// TIA Portal V21 export
// export: Created 2026-09-06T16:35:00Z, ExportSetting WithDefaults
FUNCTION "FC_LinhaCompactador_LAD" : Void   // FC21, LAD
{ S7_Optimized_Access := 'TRUE' }
VERSION : 0.1
// Visualizacao LAD da logica principal. A sequencia temporizada executavel continua em FB_LinhaCompactador.
// stored: AutoNumber true, SetENOAutomatically false
BEGIN

REGION Network 1: FC1 - OK_SISTEMA: cadeia geral de seguranca
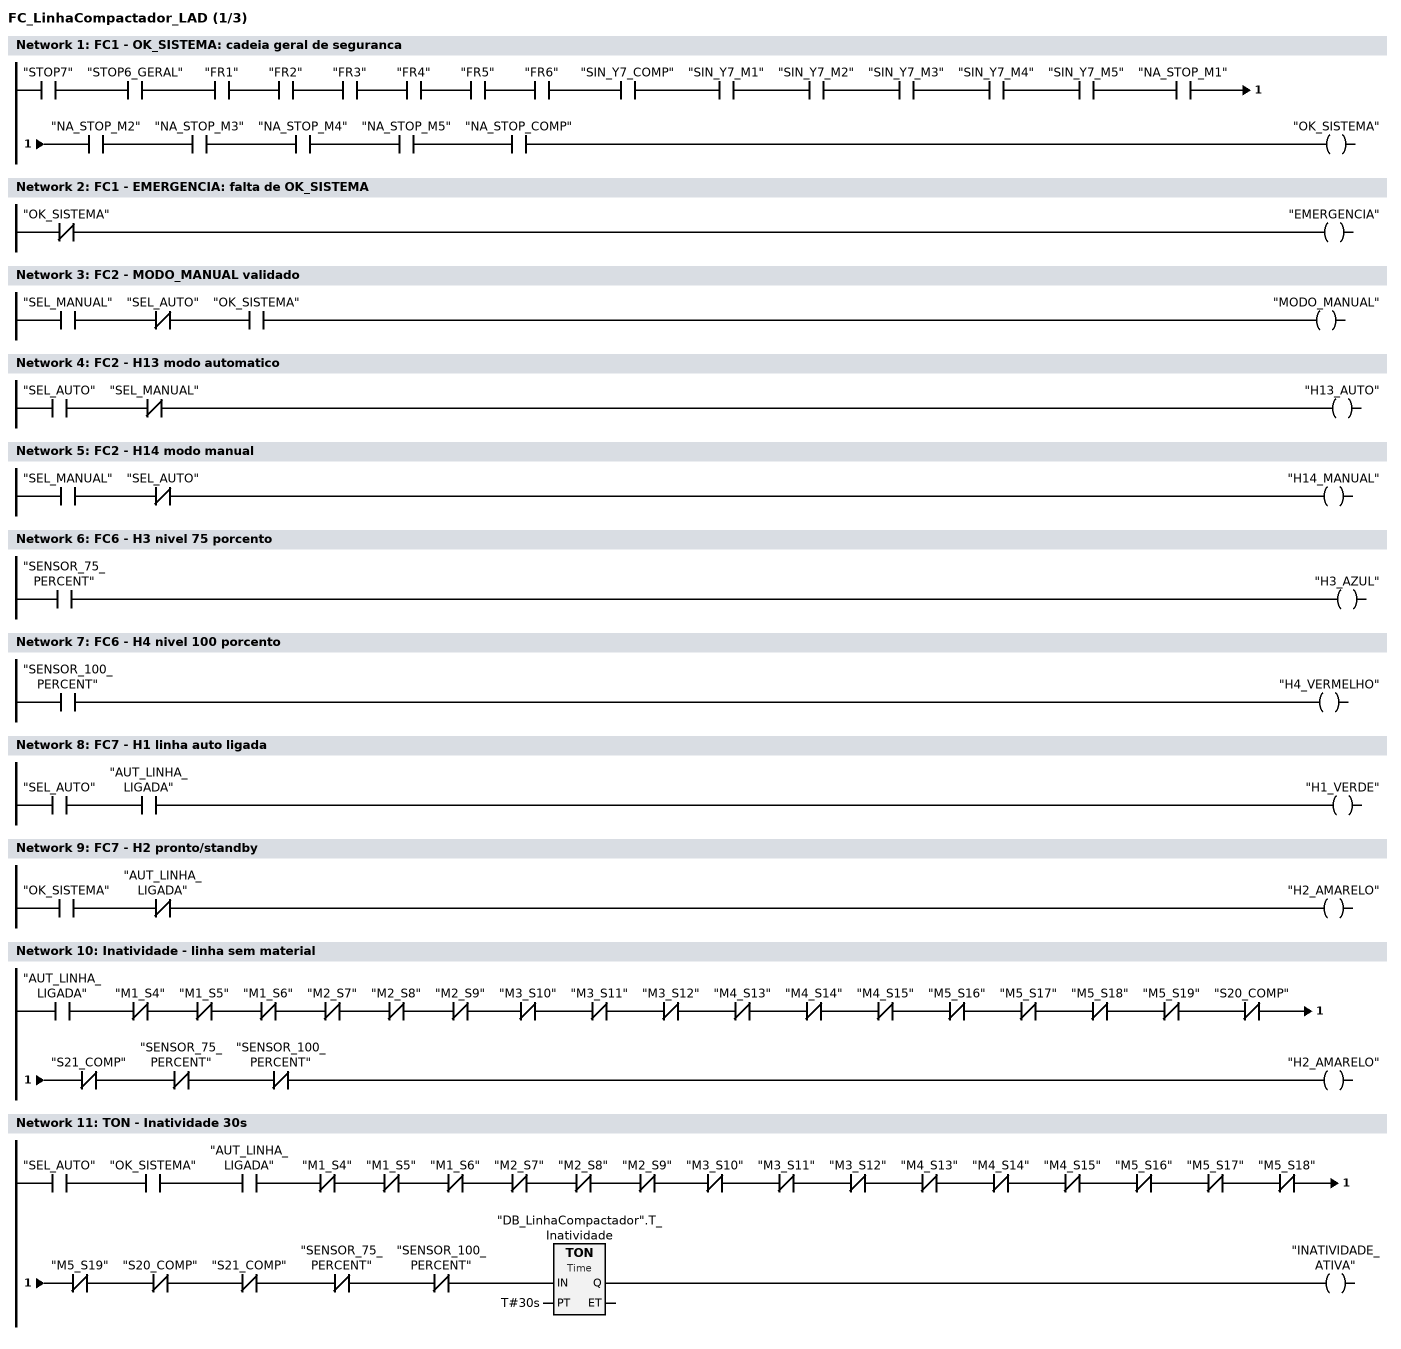
   RUNG wire#powerrail
      Contact( "STOP7" )
      Contact( "STOP6_GERAL" )
      Contact( "FR1" )
      Contact( "FR2" )
      Contact( "FR3" )
      Contact( "FR4" )
      Contact( "FR5" )
      Contact( "FR6" )
      Contact( "SIN_Y7_COMP" )
      Contact( "SIN_Y7_M1" )
      Contact( "SIN_Y7_M2" )
      Contact( "SIN_Y7_M3" )
      Contact( "SIN_Y7_M4" )
      Contact( "SIN_Y7_M5" )
      Contact( "NA_STOP_M1" )
      Contact( "NA_STOP_M2" )
      Contact( "NA_STOP_M3" )
      Contact( "NA_STOP_M4" )
      Contact( "NA_STOP_M5" )
      Contact( "NA_STOP_COMP" )
      Coil( "OK_SISTEMA" )
   END_RUNG
   // the same network as SCL:
   "OK_SISTEMA" := "STOP7" AND "STOP6_GERAL" AND "FR1" AND "FR2" AND "FR3" AND "FR4" AND "FR5" AND "FR6" AND "SIN_Y7_COMP" AND "SIN_Y7_M1" AND "SIN_Y7_M2" AND "SIN_Y7_M3" AND "SIN_Y7_M4" AND "SIN_Y7_M5" AND "NA_STOP_M1" AND "NA_STOP_M2" AND "NA_STOP_M3" AND "NA_STOP_M4" AND "NA_STOP_M5" AND "NA_STOP_COMP";
END_REGION

REGION Network 2: FC1 - EMERGENCIA: falta de OK_SISTEMA
   RUNG wire#powerrail
      I_Contact( "OK_SISTEMA" )
      Coil( "EMERGENCIA" )
   END_RUNG
   // the same network as SCL:
   "EMERGENCIA" := NOT "OK_SISTEMA";
END_REGION

REGION Network 3: FC2 - MODO_MANUAL validado
   RUNG wire#powerrail
      Contact( "SEL_MANUAL" )
      I_Contact( "SEL_AUTO" )
      Contact( "OK_SISTEMA" )
      Coil( "MODO_MANUAL" )
   END_RUNG
   // the same network as SCL:
   "MODO_MANUAL" := "SEL_MANUAL" AND NOT "SEL_AUTO" AND "OK_SISTEMA";
END_REGION

REGION Network 4: FC2 - H13 modo automatico
   RUNG wire#powerrail
      Contact( "SEL_AUTO" )
      I_Contact( "SEL_MANUAL" )
      Coil( "H13_AUTO" )
   END_RUNG
   // the same network as SCL:
   "H13_AUTO" := "SEL_AUTO" AND NOT "SEL_MANUAL";
END_REGION

REGION Network 5: FC2 - H14 modo manual
   RUNG wire#powerrail
      Contact( "SEL_MANUAL" )
      I_Contact( "SEL_AUTO" )
      Coil( "H14_MANUAL" )
   END_RUNG
   // the same network as SCL:
   "H14_MANUAL" := "SEL_MANUAL" AND NOT "SEL_AUTO";
END_REGION

REGION Network 6: FC6 - H3 nivel 75 porcento
   RUNG wire#powerrail
      Contact( "SENSOR_75_PERCENT" )
      Coil( "H3_AZUL" )
   END_RUNG
   // the same network as SCL:
   "H3_AZUL" := "SENSOR_75_PERCENT";
END_REGION

REGION Network 7: FC6 - H4 nivel 100 porcento
   RUNG wire#powerrail
      Contact( "SENSOR_100_PERCENT" )
      Coil( "H4_VERMELHO" )
   END_RUNG
   // the same network as SCL:
   "H4_VERMELHO" := "SENSOR_100_PERCENT";
END_REGION

REGION Network 8: FC7 - H1 linha auto ligada
   RUNG wire#powerrail
      Contact( "SEL_AUTO" )
      Contact( "AUT_LINHA_LIGADA" )
      Coil( "H1_VERDE" )
   END_RUNG
   // the same network as SCL:
   "H1_VERDE" := "SEL_AUTO" AND "AUT_LINHA_LIGADA";
END_REGION

REGION Network 9: FC7 - H2 pronto/standby
   RUNG wire#powerrail
      Contact( "OK_SISTEMA" )
      I_Contact( "AUT_LINHA_LIGADA" )
      Coil( "H2_AMARELO" )
   END_RUNG
   // the same network as SCL:
   "H2_AMARELO" := "OK_SISTEMA" AND NOT "AUT_LINHA_LIGADA";
END_REGION

REGION Network 10: Inatividade - linha sem material
   RUNG wire#powerrail
      Contact( "AUT_LINHA_LIGADA" )
      I_Contact( "M1_S4" )
      I_Contact( "M1_S5" )
      I_Contact( "M1_S6" )
      I_Contact( "M2_S7" )
      I_Contact( "M2_S8" )
      I_Contact( "M2_S9" )
      I_Contact( "M3_S10" )
      I_Contact( "M3_S11" )
      I_Contact( "M3_S12" )
      I_Contact( "M4_S13" )
      I_Contact( "M4_S14" )
      I_Contact( "M4_S15" )
      I_Contact( "M5_S16" )
      I_Contact( "M5_S17" )
      I_Contact( "M5_S18" )
      I_Contact( "M5_S19" )
      I_Contact( "S20_COMP" )
      I_Contact( "S21_COMP" )
      I_Contact( "SENSOR_75_PERCENT" )
      I_Contact( "SENSOR_100_PERCENT" )
      Coil( "H2_AMARELO" )
   END_RUNG
   // the same network as SCL:
   "H2_AMARELO" := "AUT_LINHA_LIGADA" AND NOT "M1_S4" AND NOT "M1_S5" AND NOT "M1_S6" AND NOT "M2_S7" AND NOT "M2_S8" AND NOT "M2_S9" AND NOT "M3_S10" AND NOT "M3_S11" AND NOT "M3_S12" AND NOT "M4_S13" AND NOT "M4_S14" AND NOT "M4_S15" AND NOT "M5_S16" AND NOT "M5_S17" AND NOT "M5_S18" AND NOT "M5_S19" AND NOT "S20_COMP" AND NOT "S21_COMP" AND NOT "SENSOR_75_PERCENT" AND NOT "SENSOR_100_PERCENT";
END_REGION

REGION Network 11: TON - Inatividade 30s
   RUNG wire#powerrail
      Contact( "SEL_AUTO" )
      Contact( "OK_SISTEMA" )
      Contact( "AUT_LINHA_LIGADA" )
      I_Contact( "M1_S4" )
      I_Contact( "M1_S5" )
      I_Contact( "M1_S6" )
      I_Contact( "M2_S7" )
      I_Contact( "M2_S8" )
      I_Contact( "M2_S9" )
      I_Contact( "M3_S10" )
      I_Contact( "M3_S11" )
      I_Contact( "M3_S12" )
      I_Contact( "M4_S13" )
      I_Contact( "M4_S14" )
      I_Contact( "M4_S15" )
      I_Contact( "M5_S16" )
      I_Contact( "M5_S17" )
      I_Contact( "M5_S18" )
      I_Contact( "M5_S19" )
      I_Contact( "S20_COMP" )
      I_Contact( "S21_COMP" )
      I_Contact( "SENSOR_75_PERCENT" )
      I_Contact( "SENSOR_100_PERCENT" )
      { S7_Templates := "time_type := Time" } "DB_LinhaCompactador".T_Inatividade.TON(pt := T#30s, et =>)
      Coil( "INATIVIDADE_ATIVA" )
   END_RUNG
   // the same network as SCL:
   "DB_LinhaCompactador".T_Inatividade.TON(IN := "SEL_AUTO" AND "OK_SISTEMA" AND "AUT_LINHA_LIGADA" AND NOT "M1_S4" AND NOT "M1_S5" AND NOT "M1_S6" AND NOT "M2_S7" AND NOT "M2_S8" AND NOT "M2_S9" AND NOT "M3_S10" AND NOT "M3_S11" AND NOT "M3_S12" AND NOT "M4_S13" AND NOT "M4_S14" AND NOT "M4_S15" AND NOT "M5_S16" AND NOT "M5_S17" AND NOT "M5_S18" AND NOT "M5_S19" AND NOT "S20_COMP" AND NOT "S21_COMP" AND NOT "SENSOR_75_PERCENT" AND NOT "SENSOR_100_PERCENT",
                           PT := T#30s);
   "INATIVIDADE_ATIVA" := "DB_LinhaCompactador".T_Inatividade.Q;
END_REGION

REGION Network 12: Manual - avanco cilindro
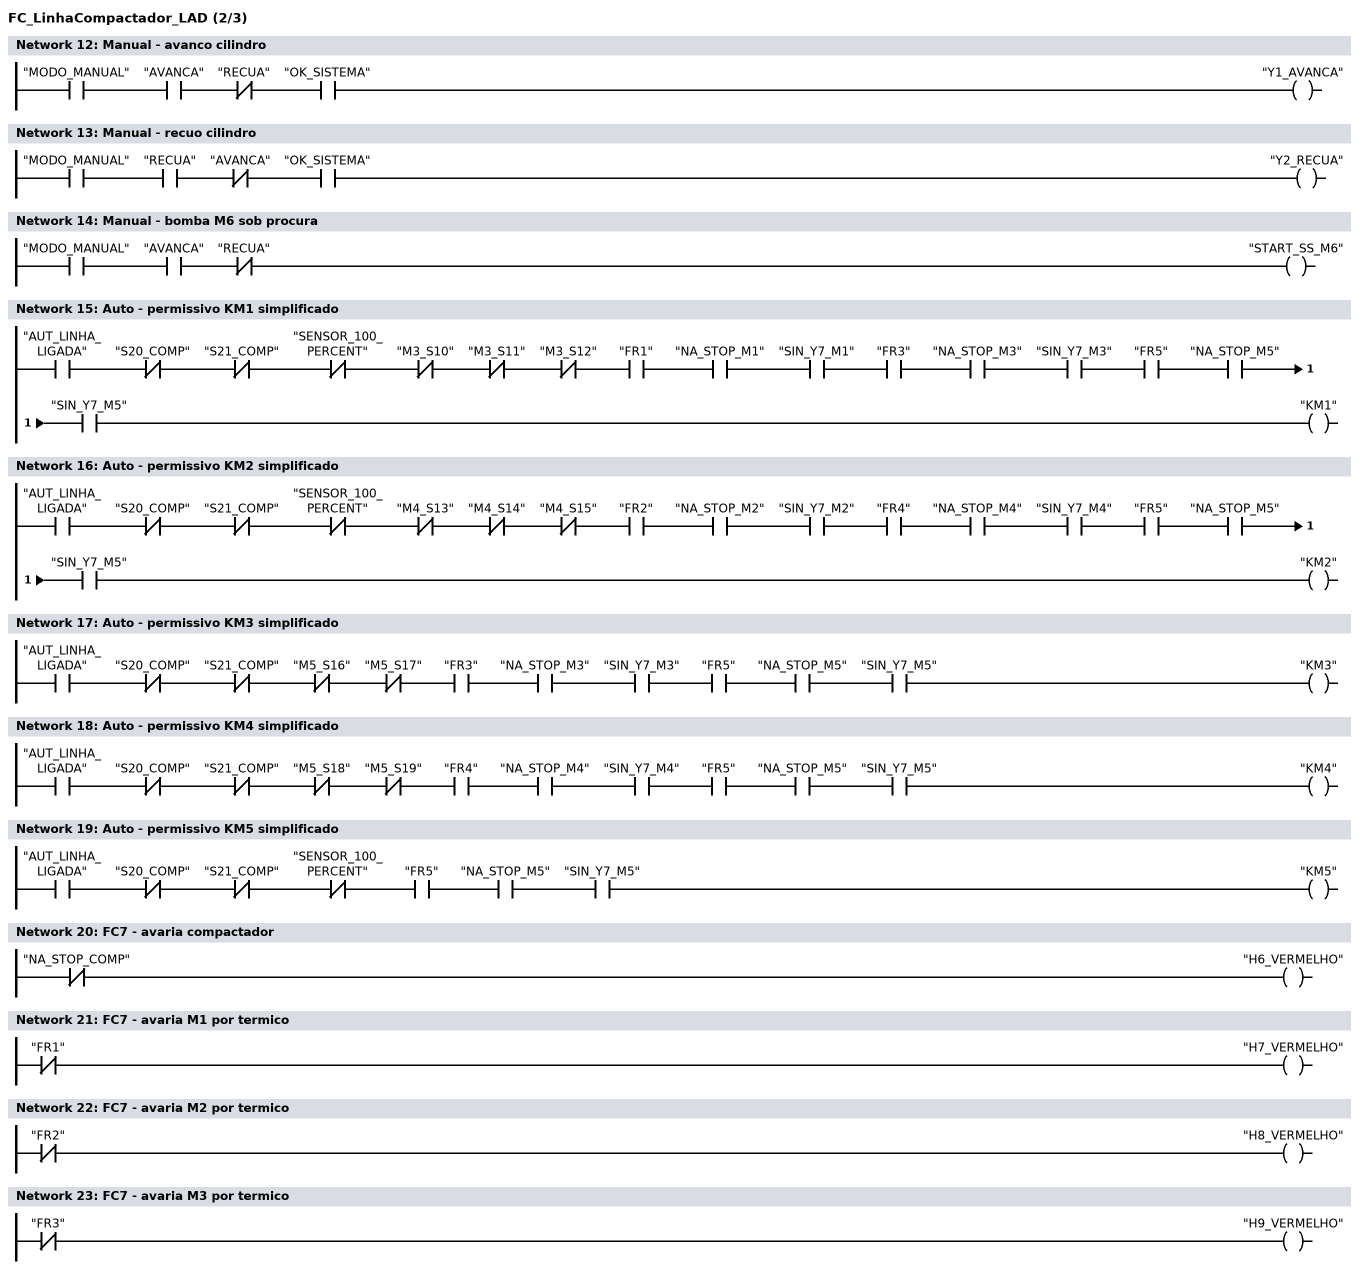
   RUNG wire#powerrail
      Contact( "MODO_MANUAL" )
      Contact( "AVANCA" )
      I_Contact( "RECUA" )
      Contact( "OK_SISTEMA" )
      Coil( "Y1_AVANCA" )
   END_RUNG
   // the same network as SCL:
   "Y1_AVANCA" := "MODO_MANUAL" AND "AVANCA" AND NOT "RECUA" AND "OK_SISTEMA";
END_REGION

REGION Network 13: Manual - recuo cilindro
   RUNG wire#powerrail
      Contact( "MODO_MANUAL" )
      Contact( "RECUA" )
      I_Contact( "AVANCA" )
      Contact( "OK_SISTEMA" )
      Coil( "Y2_RECUA" )
   END_RUNG
   // the same network as SCL:
   "Y2_RECUA" := "MODO_MANUAL" AND "RECUA" AND NOT "AVANCA" AND "OK_SISTEMA";
END_REGION

REGION Network 14: Manual - bomba M6 sob procura
   RUNG wire#powerrail
      Contact( "MODO_MANUAL" )
      Contact( "AVANCA" )
      I_Contact( "RECUA" )
      Coil( "START_SS_M6" )
   END_RUNG
   // the same network as SCL:
   "START_SS_M6" := "MODO_MANUAL" AND "AVANCA" AND NOT "RECUA";
END_REGION

REGION Network 15: Auto - permissivo KM1 simplificado
   RUNG wire#powerrail
      Contact( "AUT_LINHA_LIGADA" )
      I_Contact( "S20_COMP" )
      I_Contact( "S21_COMP" )
      I_Contact( "SENSOR_100_PERCENT" )
      I_Contact( "M3_S10" )
      I_Contact( "M3_S11" )
      I_Contact( "M3_S12" )
      Contact( "FR1" )
      Contact( "NA_STOP_M1" )
      Contact( "SIN_Y7_M1" )
      Contact( "FR3" )
      Contact( "NA_STOP_M3" )
      Contact( "SIN_Y7_M3" )
      Contact( "FR5" )
      Contact( "NA_STOP_M5" )
      Contact( "SIN_Y7_M5" )
      Coil( "KM1" )
   END_RUNG
   // the same network as SCL:
   "KM1" := "AUT_LINHA_LIGADA" AND NOT "S20_COMP" AND NOT "S21_COMP" AND NOT "SENSOR_100_PERCENT" AND NOT "M3_S10" AND NOT "M3_S11" AND NOT "M3_S12" AND "FR1" AND "NA_STOP_M1" AND "SIN_Y7_M1" AND "FR3" AND "NA_STOP_M3" AND "SIN_Y7_M3" AND "FR5" AND "NA_STOP_M5" AND "SIN_Y7_M5";
END_REGION

REGION Network 16: Auto - permissivo KM2 simplificado
   RUNG wire#powerrail
      Contact( "AUT_LINHA_LIGADA" )
      I_Contact( "S20_COMP" )
      I_Contact( "S21_COMP" )
      I_Contact( "SENSOR_100_PERCENT" )
      I_Contact( "M4_S13" )
      I_Contact( "M4_S14" )
      I_Contact( "M4_S15" )
      Contact( "FR2" )
      Contact( "NA_STOP_M2" )
      Contact( "SIN_Y7_M2" )
      Contact( "FR4" )
      Contact( "NA_STOP_M4" )
      Contact( "SIN_Y7_M4" )
      Contact( "FR5" )
      Contact( "NA_STOP_M5" )
      Contact( "SIN_Y7_M5" )
      Coil( "KM2" )
   END_RUNG
   // the same network as SCL:
   "KM2" := "AUT_LINHA_LIGADA" AND NOT "S20_COMP" AND NOT "S21_COMP" AND NOT "SENSOR_100_PERCENT" AND NOT "M4_S13" AND NOT "M4_S14" AND NOT "M4_S15" AND "FR2" AND "NA_STOP_M2" AND "SIN_Y7_M2" AND "FR4" AND "NA_STOP_M4" AND "SIN_Y7_M4" AND "FR5" AND "NA_STOP_M5" AND "SIN_Y7_M5";
END_REGION

REGION Network 17: Auto - permissivo KM3 simplificado
   RUNG wire#powerrail
      Contact( "AUT_LINHA_LIGADA" )
      I_Contact( "S20_COMP" )
      I_Contact( "S21_COMP" )
      I_Contact( "M5_S16" )
      I_Contact( "M5_S17" )
      Contact( "FR3" )
      Contact( "NA_STOP_M3" )
      Contact( "SIN_Y7_M3" )
      Contact( "FR5" )
      Contact( "NA_STOP_M5" )
      Contact( "SIN_Y7_M5" )
      Coil( "KM3" )
   END_RUNG
   // the same network as SCL:
   "KM3" := "AUT_LINHA_LIGADA" AND NOT "S20_COMP" AND NOT "S21_COMP" AND NOT "M5_S16" AND NOT "M5_S17" AND "FR3" AND "NA_STOP_M3" AND "SIN_Y7_M3" AND "FR5" AND "NA_STOP_M5" AND "SIN_Y7_M5";
END_REGION

REGION Network 18: Auto - permissivo KM4 simplificado
   RUNG wire#powerrail
      Contact( "AUT_LINHA_LIGADA" )
      I_Contact( "S20_COMP" )
      I_Contact( "S21_COMP" )
      I_Contact( "M5_S18" )
      I_Contact( "M5_S19" )
      Contact( "FR4" )
      Contact( "NA_STOP_M4" )
      Contact( "SIN_Y7_M4" )
      Contact( "FR5" )
      Contact( "NA_STOP_M5" )
      Contact( "SIN_Y7_M5" )
      Coil( "KM4" )
   END_RUNG
   // the same network as SCL:
   "KM4" := "AUT_LINHA_LIGADA" AND NOT "S20_COMP" AND NOT "S21_COMP" AND NOT "M5_S18" AND NOT "M5_S19" AND "FR4" AND "NA_STOP_M4" AND "SIN_Y7_M4" AND "FR5" AND "NA_STOP_M5" AND "SIN_Y7_M5";
END_REGION

REGION Network 19: Auto - permissivo KM5 simplificado
   RUNG wire#powerrail
      Contact( "AUT_LINHA_LIGADA" )
      I_Contact( "S20_COMP" )
      I_Contact( "S21_COMP" )
      I_Contact( "SENSOR_100_PERCENT" )
      Contact( "FR5" )
      Contact( "NA_STOP_M5" )
      Contact( "SIN_Y7_M5" )
      Coil( "KM5" )
   END_RUNG
   // the same network as SCL:
   "KM5" := "AUT_LINHA_LIGADA" AND NOT "S20_COMP" AND NOT "S21_COMP" AND NOT "SENSOR_100_PERCENT" AND "FR5" AND "NA_STOP_M5" AND "SIN_Y7_M5";
END_REGION

REGION Network 20: FC7 - avaria compactador
   RUNG wire#powerrail
      I_Contact( "NA_STOP_COMP" )
      Coil( "H6_VERMELHO" )
   END_RUNG
   // the same network as SCL:
   "H6_VERMELHO" := NOT "NA_STOP_COMP";
END_REGION

REGION Network 21: FC7 - avaria M1 por termico
   RUNG wire#powerrail
      I_Contact( "FR1" )
      Coil( "H7_VERMELHO" )
   END_RUNG
   // the same network as SCL:
   "H7_VERMELHO" := NOT "FR1";
END_REGION

REGION Network 22: FC7 - avaria M2 por termico
   RUNG wire#powerrail
      I_Contact( "FR2" )
      Coil( "H8_VERMELHO" )
   END_RUNG
   // the same network as SCL:
   "H8_VERMELHO" := NOT "FR2";
END_REGION

REGION Network 23: FC7 - avaria M3 por termico
   RUNG wire#powerrail
      I_Contact( "FR3" )
      Coil( "H9_VERMELHO" )
   END_RUNG
   // the same network as SCL:
   "H9_VERMELHO" := NOT "FR3";
END_REGION

REGION Network 24: FC7 - avaria M4 por termico
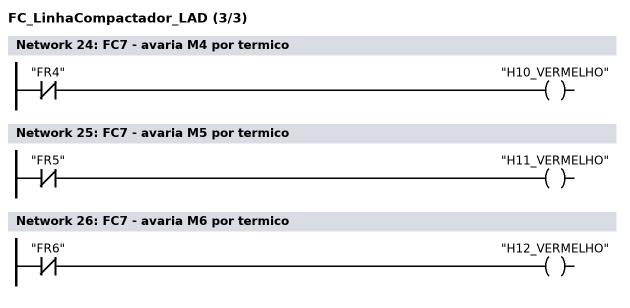
   RUNG wire#powerrail
      I_Contact( "FR4" )
      Coil( "H10_VERMELHO" )
   END_RUNG
   // the same network as SCL:
   "H10_VERMELHO" := NOT "FR4";
END_REGION

REGION Network 25: FC7 - avaria M5 por termico
   RUNG wire#powerrail
      I_Contact( "FR5" )
      Coil( "H11_VERMELHO" )
   END_RUNG
   // the same network as SCL:
   "H11_VERMELHO" := NOT "FR5";
END_REGION

REGION Network 26: FC7 - avaria M6 por termico
   RUNG wire#powerrail
      I_Contact( "FR6" )
      Coil( "H12_VERMELHO" )
   END_RUNG
   // the same network as SCL:
   "H12_VERMELHO" := NOT "FR6";
END_REGION
END_FUNCTION
